{attribute 'qualified_only'}

TYPE inserterUnLoadDisplayStates :
(
	dStStartUp,
	dStStandBy,
	dStStationIsStopped,
	dStStationIsReseting,
	dStWorking,
	dStStationReady,
	dStWaitForNextStep,

	dStGripperDidNotClose,
	dStGripperDidNotOpen,
	dStInserterDidNotMoveDown,
	dStInserterDidNotMoveUp,
	dStDriveDidNotHome,
	dStDriveTimeOutMove,
	dStDriveError,
	dStCameraTimeOut,
	dStCameraError,
	dStCameraBadResult,
	dStInitSensorGripError,
	dStNoSensorInNest
	
	
)DINT;
END_TYPE

(* stored: Version 1.1.0.1, ProductVersion 3.1.4024.3
   DUT inserterUnLoadDisplayStates: Id {f51d7071-508d-495d-8053-f32657da31cd} *)
